SUBAPPLICATION mapping_Uebung_005 (* Toggle Flip-Flop mit IE *)
  (* Standard: 61499-2 *)
  (* Version 1.0, 2023-10-23, franz *)
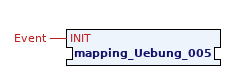
  EVENT_INPUT
    INIT;
  END_EVENT
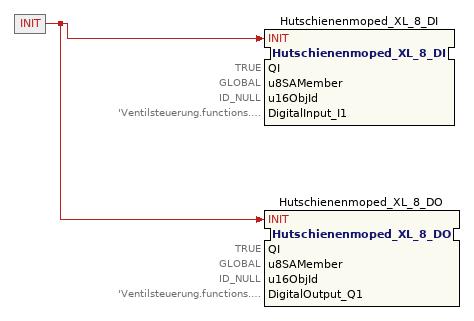
  FBS
    Hutschienenmoped_XL_8_DO : Hutschienenmoped_XL_8_DO(QI := TRUE, u8SAMember := GLOBAL, u16ObjId := ID_NULL, DigitalOutput_Q1 := 'Ventilsteuerung.functions.DigitalOutput_Q1');
    Hutschienenmoped_XL_8_DI : Hutschienenmoped_XL_8_DI(QI := TRUE, u8SAMember := GLOBAL, u16ObjId := ID_NULL, DigitalInput_I1 := 'Ventilsteuerung.functions.DigitalInput_I1');
  END_FBS
  EVENT_CONNECTIONS
    INIT TO Hutschienenmoped_XL_8_DO.INIT;
    INIT TO Hutschienenmoped_XL_8_DI.INIT;
  END_CONNECTIONS
END_SUBAPPLICATION
